TYPE ST_InverterControlWord :
STRUCT
	b_ChargeDC				: BOOL;
	b_run					: BOOL;
	b_Reset					: BOOL;
	b_FieldbusControlEnable	: BOOL;
	b_WatchdogPulse			: BOOL;
	b_ParallelAFE			: BOOL;
	b_PIDenable				: BOOL;
	b_GridCodeEnable		: BOOL;
	b_ExtGridcodeTrip		: BOOL;
END_STRUCT
END_TYPE

(* stored: Version 1.1.0.1, ProductVersion 3.1.4026.18
   DUT ST_InverterControlWord: Id {a2f5a00b-5714-4764-bfb9-c612d5f94142} *)
